FUNCTION_BLOCK CL_AxisL1LeftFront EXTENDS CL_AxisRobot
var
END_VAR

SUPER^();

METHOD PROTECTED InitDefect : BOOL
sWhichAxis := 'left(L1)-front';
InitDefect := true;
END_METHOD

END_FUNCTION_BLOCK

(* stored: Version 1.1.0.1, ProductVersion 3.1.4024.12
   POU CL_AxisL1LeftFront: Id {d5d457c4-b3f3-4d4e-906d-770cc886d557}, SpecialFunc None
   Method InitDefect: Id {5b773ca0-6402-4f85-8ced-27749da5bd34} *)
